// TIA Portal V20 export
// export: Created 2026-07-22T09:37:42.5992996Z, ExportSetting WithDefaults, DisplayName Totally Integrated Automation Portal, DisplayVersion V20, DisplayName TIA Portal Openness, DisplayVersion V20, DisplayName TIA Portal Version Control Interface, DisplayVersion V20, DisplayName STEP 7 Professional, DisplayVersion V20, DisplayName STEP 7 Safety, DisplayVersion V20, DisplayName WinCC Basic/Comfort/Advanced, DisplayVersion V20, DisplayName WinCC Professional, DisplayVersion V20, DisplayName WinCC Unified, DisplayVersion V20
FUNCTION_BLOCK "FB_ValveControl"   // FB1, LAD
{ S7_Optimized_Access := 'TRUE' }
VERSION : 0.1
// stored: AutoNumber true, IsIECCheckEnabled false, IsRetainMemResEnabled false, MemoryReserve 100, SetENOAutomatically false, UDAEnableTagReadback false
   VAR_INPUT
      OpenCmd : Bool;
      CloseCmd : Bool;
      LocalMode : Bool;
      Healthy : Bool;
      OpenFB : Bool;
      ClosedFB : Bool;
   END_VAR
   VAR_OUTPUT
      OpenValve : Bool;
      CloseValve : Bool;
   END_VAR
BEGIN

REGION Network 1
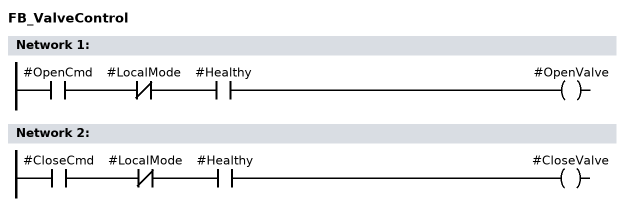
   RUNG wire#powerrail
      Contact( #OpenCmd )
      I_Contact( #LocalMode )
      Contact( #Healthy )
      Coil( #OpenValve )
   END_RUNG
   // the same network as SCL:
   #OpenValve := #OpenCmd AND NOT #LocalMode AND #Healthy;
END_REGION

REGION Network 2
   RUNG wire#powerrail
      Contact( #CloseCmd )
      I_Contact( #LocalMode )
      Contact( #Healthy )
      Coil( #CloseValve )
   END_RUNG
   // the same network as SCL:
   #CloseValve := #CloseCmd AND NOT #LocalMode AND #Healthy;
END_REGION
END_FUNCTION_BLOCK
